MoveL [[1651.97,-191.36,-511.21],[0.032971,0.999448,0.003972,-0.00071],[0,-1,-1,0],[0,9E9,9E9,9E9,9E9,9E9]],Work,z10,custom_tool1\WObj:=WObj0;
MoveL [[1651.88,-186.36,-511.2],[0.032971,0.999448,0.003972,-0.00071],[0,-1,-1,0],[0,9E9,9E9,9E9,9E9,9E9]],Work,z10,custom_tool1\WObj:=WObj0;
MoveL [[1651.8,-181.36,-511.19],[0.032971,0.999448,0.003972,-0.00071],[0,-1,-1,0],[0,9E9,9E9,9E9,9E9,9E9]],Work,z10,custom_tool1\WObj:=WObj0;
MoveL [[1651.72,-176.36,-511.19],[0.032971,0.999448,0.003972,-0.00071],[0,-1,-1,0],[0,9E9,9E9,9E9,9E9,9E9]],Work,z10,custom_tool1\WObj:=WObj0;
MoveL [[1651.64,-171.36,-511.18],[0.032971,0.999448,0.003972,-0.00071],[0,-1,-1,0],[0,9E9,9E9,9E9,9E9,9E9]],Work,z10,custom_tool1\WObj:=WObj0;
MoveL [[1651.55,-166.36,-511.17],[0.032971,0.999448,0.003972,-0.00071],[0,-1,-1,0],[0,9E9,9E9,9E9,9E9,9E9]],Work,z10,custom_tool1\WObj:=WObj0;
MoveL [[1651.47,-161.36,-511.16],[0.032971,0.999448,0.003972,-0.00071],[0,-1,-1,0],[0,9E9,9E9,9E9,9E9,9E9]],Work,z10,custom_tool1\WObj:=WObj0;
MoveL [[1651.39,-156.36,-511.16],[0.032971,0.999448,0.003972,-0.00071],[0,-1,-1,0],[0,9E9,9E9,9E9,9E9,9E9]],Work,z10,custom_tool1\WObj:=WObj0;
MoveL [[1651.31,-151.36,-511.15],[0.032971,0.999448,0.003972,-0.00071],[0,-1,-1,0],[0,9E9,9E9,9E9,9E9,9E9]],Work,z10,custom_tool1\WObj:=WObj0;
MoveL [[1650.68,-145.74,-511.14],[0.032971,0.999448,0.003972,-0.00071],[0,-1,-1,0],[0,9E9,9E9,9E9,9E9,9E9]],Work,z10,custom_tool1\WObj:=WObj0;
MoveL [[1650.05,-140.11,-511.13],[0.032971,0.999448,0.003972,-0.00071],[0,-1,-1,0],[0,9E9,9E9,9E9,9E9,9E9]],Work,z10,custom_tool1\WObj:=WObj0;
MoveL [[1648.24,-134.38,-511.12],[0.032971,0.999448,0.003972,-0.00071],[0,-1,-1,0],[0,9E9,9E9,9E9,9E9,9E9]],Work,z10,custom_tool1\WObj:=WObj0;
MoveL [[1646.43,-128.65,-511.11],[0.032971,0.999448,0.003972,-0.00071],[0,-1,-1,0],[0,9E9,9E9,9E9,9E9,9E9]],Work,z10,custom_tool1\WObj:=WObj0;
MoveL [[1643.51,-123.38,-511.1],[0.032971,0.999448,0.003972,-0.00071],[0,-1,-1,0],[0,9E9,9E9,9E9,9E9,9E9]],Work,z10,custom_tool1\WObj:=WObj0;
MoveL [[1640.59,-118.12,-511.08],[0.032971,0.999448,0.003972,-0.00071],[0,-1,-1,0],[0,9E9,9E9,9E9,9E9,9E9]],Work,z10,custom_tool1\WObj:=WObj0;
MoveL [[1636.59,-113.46,-511.07],[0.032971,0.999448,0.003972,-0.00071],[0,-1,-1,0],[0,9E9,9E9,9E9,9E9,9E9]],Work,z10,custom_tool1\WObj:=WObj0;
MoveL [[1632.58,-108.8,-511.06],[0.032971,0.999448,0.003972,-0.00071],[0,-1,-1,0],[0,9E9,9E9,9E9,9E9,9E9]],Work,z10,custom_tool1\WObj:=WObj0;
MoveL [[1627.75,-105.08,-511.04],[0.032971,0.999448,0.003972,-0.00071],[0,-1,-1,0],[0,9E9,9E9,9E9,9E9,9E9]],Work,z10,custom_tool1\WObj:=WObj0;
MoveL [[1622.92,-101.35,-511.03],[0.032971,0.999448,0.003972,-0.00071],[0,-1,-1,0],[0,9E9,9E9,9E9,9E9,9E9]],Work,z10,custom_tool1\WObj:=WObj0;
MoveL [[1617.56,-98.73,-511.01],[0.032971,0.999448,0.003972,-0.00071],[0,-1,-1,0],[0,9E9,9E9,9E9,9E9,9E9]],Work,z10,custom_tool1\WObj:=WObj0;
MoveL [[1612.2,-96.1,-511],[0.032971,0.999448,0.003972,-0.00071],[0,-1,-1,0],[0,9E9,9E9,9E9,9E9,9E9]],Work,z10,custom_tool1\WObj:=WObj0;
MoveL [[1606.66,-94.63,-510.98],[0.032971,0.999448,0.003972,-0.00071],[0,-1,-1,0],[0,9E9,9E9,9E9,9E9,9E9]],Work,z10,custom_tool1\WObj:=WObj0;
MoveL [[1601.12,-93.16,-510.97],[0.032971,0.999448,0.003972,-0.00071],[0,-1,-1,0],[0,9E9,9E9,9E9,9E9,9E9]],Work,z10,custom_tool1\WObj:=WObj0;
MoveL [[1595.72,-92.76,-510.96],[0.032971,0.999448,0.003972,-0.00071],[0,-1,-1,0],[0,9E9,9E9,9E9,9E9,9E9]],Work,z10,custom_tool1\WObj:=WObj0;
MoveL [[1590.33,-92.36,-510.95],[0.032971,0.999448,0.003972,-0.00071],[0,-1,-1,0],[0,9E9,9E9,9E9,9E9,9E9]],Work,z10,custom_tool1\WObj:=WObj0;
MoveL [[1585.16,-92.45,-510.94],[0.032971,0.999448,0.003972,-0.00071],[0,-1,-1,0],[0,9E9,9E9,9E9,9E9,9E9]],Work,z10,custom_tool1\WObj:=WObj0;
MoveL [[1579.99,-92.53,-510.93],[0.032971,0.999448,0.003972,-0.00071],[0,-1,-1,0],[0,9E9,9E9,9E9,9E9,9E9]],Work,z10,custom_tool1\WObj:=WObj0;
MoveL [[1574.83,-92.62,-510.92],[0.032971,0.999448,0.003972,-0.00071],[0,-1,-1,0],[0,9E9,9E9,9E9,9E9,9E9]],Work,z10,custom_tool1\WObj:=WObj0;
MoveL [[1569.66,-92.7,-510.91],[0.032971,0.999448,0.003972,-0.00071],[0,-1,-1,0],[0,9E9,9E9,9E9,9E9,9E9]],Work,z10,custom_tool1\WObj:=WObj0;
MoveL [[1564.5,-92.79,-510.9],[0.032971,0.999448,0.003972,-0.00071],[0,-1,-1,0],[0,9E9,9E9,9E9,9E9,9E9]],Work,z10,custom_tool1\WObj:=WObj0;
MoveL [[1559.33,-92.87,-510.89],[0.032971,0.999448,0.003972,-0.00071],[0,-1,-1,0],[0,9E9,9E9,9E9,9E9,9E9]],Work,z10,custom_tool1\WObj:=WObj0;
MoveL [[1554.16,-92.96,-510.88],[0.032971,0.999448,0.003972,-0.00071],[0,-1,-1,0],[0,9E9,9E9,9E9,9E9,9E9]],Work,z10,custom_tool1\WObj:=WObj0;
MoveL [[1549,-93.04,-510.87],[0.032971,0.999448,0.003972,-0.00071],[0,-1,-1,0],[0,9E9,9E9,9E9,9E9,9E9]],Work,z10,custom_tool1\WObj:=WObj0;
MoveL [[1543.83,-93.13,-510.86],[0.032971,0.999448,0.003972,-0.00071],[0,-1,-1,0],[0,9E9,9E9,9E9,9E9,9E9]],Work,z10,custom_tool1\WObj:=WObj0;
MoveL [[1538.67,-93.21,-510.85],[0.032971,0.999448,0.003972,-0.00071],[0,-1,-1,0],[0,9E9,9E9,9E9,9E9,9E9]],Work,z10,custom_tool1\WObj:=WObj0;
MoveL [[1533.5,-93.3,-510.84],[0.032971,0.999448,0.003972,-0.00071],[0,-1,-1,0],[0,9E9,9E9,9E9,9E9,9E9]],Work,z10,custom_tool1\WObj:=WObj0;
MoveL [[1528.33,-93.38,-510.83],[0.032971,0.999448,0.003972,-0.00071],[0,-1,-1,0],[0,9E9,9E9,9E9,9E9,9E9]],Work,z10,custom_tool1\WObj:=WObj0;
MoveL [[1523.41,-94.44,-510.82],[0.032971,0.999448,0.003972,-0.00071],[0,-1,-1,0],[0,9E9,9E9,9E9,9E9,9E9]],Work,z10,custom_tool1\WObj:=WObj0;
MoveL [[1518.49,-95.49,-510.81],[0.032971,0.999448,0.003972,-0.00071],[0,-1,-1,0],[0,9E9,9E9,9E9,9E9,9E9]],Work,z10,custom_tool1\WObj:=WObj0;
MoveL [[1513.57,-96.55,-510.8],[0.032971,0.999448,0.003972,-0.00071],[0,-1,-1,0],[0,9E9,9E9,9E9,9E9,9E9]],Work,z10,custom_tool1\WObj:=WObj0;
MoveL [[1508.65,-97.61,-510.79],[0.032971,0.999448,0.003972,-0.00071],[0,-1,-1,0],[0,9E9,9E9,9E9,9E9,9E9]],Work,z10,custom_tool1\WObj:=WObj0;
MoveL [[1505.66,-98.24,-510.79],[0.032971,0.999448,0.003972,-0.00071],[0,-1,-1,0],[0,9E9,9E9,9E9,9E9,9E9]],Work,z10,custom_tool1\WObj:=WObj0;
MoveL [[1501.69,-101,-510.78],[0.032971,0.999448,0.003972,-0.00071],[0,-1,-1,0],[0,9E9,9E9,9E9,9E9,9E9]],Work,z10,custom_tool1\WObj:=WObj0;
MoveL [[1497.72,-103.77,-510.78],[0.032971,0.999448,0.003972,-0.00071],[0,-1,-1,0],[0,9E9,9E9,9E9,9E9,9E9]],Work,z10,custom_tool1\WObj:=WObj0;
MoveL [[1493.75,-106.54,-510.78],[0.032971,0.999448,0.003972,-0.00071],[0,-1,-1,0],[0,9E9,9E9,9E9,9E9,9E9]],Work,z10,custom_tool1\WObj:=WObj0;
MoveL [[1489.77,-109.31,-510.77],[0.032971,0.999448,0.003972,-0.00071],[0,-1,-1,0],[0,9E9,9E9,9E9,9E9,9E9]],Work,z10,custom_tool1\WObj:=WObj0;
MoveL [[1485.8,-112.07,-510.77],[0.032971,0.999448,0.003972,-0.00071],[0,-1,-1,0],[0,9E9,9E9,9E9,9E9,9E9]],Work,z10,custom_tool1\WObj:=WObj0;
MoveL [[1483.26,-116.15,-510.77],[0.032971,0.999448,0.003972,-0.00071],[0,-1,-1,0],[0,9E9,9E9,9E9,9E9,9E9]],Work,z10,custom_tool1\WObj:=WObj0;
MoveL [[1480.71,-120.23,-510.77],[0.032971,0.999448,0.003972,-0.00071],[0,-1,-1,0],[0,9E9,9E9,9E9,9E9,9E9]],Work,z10,custom_tool1\WObj:=WObj0;
MoveL [[1478.17,-124.31,-510.77],[0.032971,0.999448,0.003972,-0.00071],[0,-1,-1,0],[0,9E9,9E9,9E9,9E9,9E9]],Work,z10,custom_tool1\WObj:=WObj0;
MoveL [[1475.63,-128.39,-510.77],[0.032971,0.999448,0.003972,-0.00071],[0,-1,-1,0],[0,9E9,9E9,9E9,9E9,9E9]],Work,z10,custom_tool1\WObj:=WObj0;
MoveL [[1473.08,-132.47,-510.77],[0.032971,0.999448,0.003972,-0.00071],[0,-1,-1,0],[0,9E9,9E9,9E9,9E9,9E9]],Work,z10,custom_tool1\WObj:=WObj0;
MoveL [[1472.58,-135.41,-510.77],[0.032971,0.999448,0.003972,-0.00071],[0,-1,-1,0],[0,9E9,9E9,9E9,9E9,9E9]],Work,z10,custom_tool1\WObj:=WObj0;
MoveL [[1471.76,-140.15,-510.78],[0.032971,0.999448,0.003972,-0.00071],[0,-1,-1,0],[0,9E9,9E9,9E9,9E9,9E9]],Work,z10,custom_tool1\WObj:=WObj0;
MoveL [[1470.95,-144.89,-510.78],[0.032971,0.999448,0.003972,-0.00071],[0,-1,-1,0],[0,9E9,9E9,9E9,9E9,9E9]],Work,z10,custom_tool1\WObj:=WObj0;
MoveL [[1470.14,-149.63,-510.79],[0.032971,0.999448,0.003972,-0.00071],[0,-1,-1,0],[0,9E9,9E9,9E9,9E9,9E9]],Work,z10,custom_tool1\WObj:=WObj0;
MoveL [[1469.33,-154.36,-510.79],[0.032971,0.999448,0.003972,-0.00071],[0,-1,-1,0],[0,9E9,9E9,9E9,9E9,9E9]],Work,z10,custom_tool1\WObj:=WObj0;
MoveL [[1469.41,-159.35,-510.8],[0.032971,0.999448,0.003972,-0.00071],[0,-1,-1,0],[0,9E9,9E9,9E9,9E9,9E9]],Work,z10,custom_tool1\WObj:=WObj0;
MoveL [[1469.5,-164.33,-510.81],[0.032971,0.999448,0.003972,-0.00071],[0,-1,-1,0],[0,9E9,9E9,9E9,9E9,9E9]],Work,z10,custom_tool1\WObj:=WObj0;
MoveL [[1469.58,-169.31,-510.81],[0.032971,0.999448,0.003972,-0.00071],[0,-1,-1,0],[0,9E9,9E9,9E9,9E9,9E9]],Work,z10,custom_tool1\WObj:=WObj0;
MoveL [[1469.66,-174.29,-510.82],[0.032971,0.999448,0.003972,-0.00071],[0,-1,-1,0],[0,9E9,9E9,9E9,9E9,9E9]],Work,z10,custom_tool1\WObj:=WObj0;
MoveL [[1469.74,-179.28,-510.83],[0.032971,0.999448,0.003972,-0.00071],[0,-1,-1,0],[0,9E9,9E9,9E9,9E9,9E9]],Work,z10,custom_tool1\WObj:=WObj0;
MoveL [[1469.82,-184.26,-510.83],[0.032971,0.999448,0.003972,-0.00071],[0,-1,-1,0],[0,9E9,9E9,9E9,9E9,9E9]],Work,z10,custom_tool1\WObj:=WObj0;
MoveL [[1469.91,-189.24,-510.84],[0.032971,0.999448,0.003972,-0.00071],[0,-1,-1,0],[0,9E9,9E9,9E9,9E9,9E9]],Work,z10,custom_tool1\WObj:=WObj0;
MoveL [[1469.99,-194.23,-510.85],[0.032971,0.999448,0.003972,-0.00071],[0,-1,-1,0],[0,9E9,9E9,9E9,9E9,9E9]],Work,z10,custom_tool1\WObj:=WObj0;
MoveL [[1470.07,-199.21,-510.85],[0.032971,0.999448,0.003972,-0.00071],[0,-1,-1,0],[0,9E9,9E9,9E9,9E9,9E9]],Work,z10,custom_tool1\WObj:=WObj0;
MoveL [[1470.15,-204.19,-510.86],[0.032971,0.999448,0.003972,-0.00071],[0,-1,-1,0],[0,9E9,9E9,9E9,9E9,9E9]],Work,z10,custom_tool1\WObj:=WObj0;
MoveL [[1470.24,-209.17,-510.87],[0.032971,0.999448,0.003972,-0.00071],[0,-1,-1,0],[0,9E9,9E9,9E9,9E9,9E9]],Work,z10,custom_tool1\WObj:=WObj0;
MoveL [[1470.32,-214.16,-510.88],[0.032971,0.999448,0.003972,-0.00071],[0,-1,-1,0],[0,9E9,9E9,9E9,9E9,9E9]],Work,z10,custom_tool1\WObj:=WObj0;
MoveL [[1470.4,-219.14,-510.88],[0.032971,0.999448,0.003972,-0.00071],[0,-1,-1,0],[0,9E9,9E9,9E9,9E9,9E9]],Work,z10,custom_tool1\WObj:=WObj0;
MoveL [[1470.48,-224.12,-510.89],[0.032971,0.999448,0.003972,-0.00071],[0,-1,-1,0],[0,9E9,9E9,9E9,9E9,9E9]],Work,z10,custom_tool1\WObj:=WObj0;
MoveL [[1470.56,-229.1,-510.9],[0.032971,0.999448,0.003972,-0.00071],[0,-1,-1,0],[0,9E9,9E9,9E9,9E9,9E9]],Work,z10,custom_tool1\WObj:=WObj0;
MoveL [[1470.65,-234.09,-510.9],[0.032971,0.999448,0.003972,-0.00071],[0,-1,-1,0],[0,9E9,9E9,9E9,9E9,9E9]],Work,z10,custom_tool1\WObj:=WObj0;
MoveL [[1470.73,-239.07,-510.91],[0.032971,0.999448,0.003972,-0.00071],[0,-1,-1,0],[0,9E9,9E9,9E9,9E9,9E9]],Work,z10,custom_tool1\WObj:=WObj0;
MoveL [[1470.81,-244.05,-510.92],[0.032971,0.999448,0.003972,-0.00071],[0,-1,-1,0],[0,9E9,9E9,9E9,9E9,9E9]],Work,z10,custom_tool1\WObj:=WObj0;
MoveL [[1470.89,-249.03,-510.92],[0.032971,0.999448,0.003972,-0.00071],[0,-1,-1,0],[0,9E9,9E9,9E9,9E9,9E9]],Work,z10,custom_tool1\WObj:=WObj0;
MoveL [[1470.97,-254.02,-510.93],[0.032971,0.999448,0.003972,-0.00071],[0,-1,-1,0],[0,9E9,9E9,9E9,9E9,9E9]],Work,z10,custom_tool1\WObj:=WObj0;
MoveL [[1471.06,-259.13,-510.94],[0.032971,0.999448,0.003972,-0.00071],[0,-1,-1,0],[0,9E9,9E9,9E9,9E9,9E9]],Work,z10,custom_tool1\WObj:=WObj0;
MoveL [[1471.14,-264.24,-510.94],[0.032971,0.999448,0.003972,-0.00071],[0,-1,-1,0],[0,9E9,9E9,9E9,9E9,9E9]],Work,z10,custom_tool1\WObj:=WObj0;
MoveL [[1471.23,-269.35,-510.95],[0.032971,0.999448,0.003972,-0.00071],[0,-1,-1,0],[0,9E9,9E9,9E9,9E9,9E9]],Work,z10,custom_tool1\WObj:=WObj0;
MoveL [[1471.31,-274.46,-510.96],[0.032971,0.999448,0.003972,-0.00071],[0,-1,-1,0],[0,9E9,9E9,9E9,9E9,9E9]],Work,z10,custom_tool1\WObj:=WObj0;
MoveL [[1471.4,-279.57,-510.97],[0.032971,0.999448,0.003972,-0.00071],[0,-1,-1,0],[0,9E9,9E9,9E9,9E9,9E9]],Work,z10,custom_tool1\WObj:=WObj0;
MoveL [[1471.48,-284.68,-510.97],[0.032971,0.999448,0.003972,-0.00071],[0,-1,-1,0],[0,9E9,9E9,9E9,9E9,9E9]],Work,z10,custom_tool1\WObj:=WObj0;
MoveL [[1471.56,-289.66,-510.98],[0.032971,0.999448,0.003972,-0.00071],[0,-1,-1,0],[0,9E9,9E9,9E9,9E9,9E9]],Work,z10,custom_tool1\WObj:=WObj0;
MoveL [[1471.64,-294.64,-510.99],[0.032971,0.999448,0.003972,-0.00071],[0,-1,-1,0],[0,9E9,9E9,9E9,9E9,9E9]],Work,z10,custom_tool1\WObj:=WObj0;
MoveL [[1471.73,-299.63,-510.99],[0.032971,0.999448,0.003972,-0.00071],[0,-1,-1,0],[0,9E9,9E9,9E9,9E9,9E9]],Work,z10,custom_tool1\WObj:=WObj0;
MoveL [[1471.81,-304.61,-511],[0.032971,0.999448,0.003972,-0.00071],[0,-1,-1,0],[0,9E9,9E9,9E9,9E9,9E9]],Work,z10,custom_tool1\WObj:=WObj0;
MoveL [[1471.89,-309.59,-511.01],[0.032971,0.999448,0.003972,-0.00071],[0,-1,-1,0],[0,9E9,9E9,9E9,9E9,9E9]],Work,z10,custom_tool1\WObj:=WObj0;
MoveL [[1471.97,-314.58,-511.01],[0.032971,0.999448,0.003972,-0.00071],[0,-1,-1,0],[0,9E9,9E9,9E9,9E9,9E9]],Work,z10,custom_tool1\WObj:=WObj0;
MoveL [[1472.06,-319.56,-511.02],[0.032971,0.999448,0.003972,-0.00071],[0,-1,-1,0],[0,9E9,9E9,9E9,9E9,9E9]],Work,z10,custom_tool1\WObj:=WObj0;
MoveL [[1472.14,-324.54,-511.03],[0.032971,0.999448,0.003972,-0.00071],[0,-1,-1,0],[0,9E9,9E9,9E9,9E9,9E9]],Work,z10,custom_tool1\WObj:=WObj0;
MoveL [[1472.22,-329.52,-511.04],[0.032971,0.999448,0.003972,-0.00071],[0,-1,-1,0],[0,9E9,9E9,9E9,9E9,9E9]],Work,z10,custom_tool1\WObj:=WObj0;
MoveL [[1472.3,-334.51,-511.04],[0.032971,0.999448,0.003972,-0.00071],[0,-1,-1,0],[0,9E9,9E9,9E9,9E9,9E9]],Work,z10,custom_tool1\WObj:=WObj0;
MoveL [[1472.38,-339.49,-511.05],[0.032971,0.999448,0.003972,-0.00071],[0,-1,-1,0],[0,9E9,9E9,9E9,9E9,9E9]],Work,z10,custom_tool1\WObj:=WObj0;
MoveL [[1472.47,-344.47,-511.06],[0.032971,0.999448,0.003972,-0.00071],[0,-1,-1,0],[0,9E9,9E9,9E9,9E9,9E9]],Work,z10,custom_tool1\WObj:=WObj0;
MoveL [[1472.55,-349.45,-511.06],[0.032971,0.999448,0.003972,-0.00071],[0,-1,-1,0],[0,9E9,9E9,9E9,9E9,9E9]],Work,z10,custom_tool1\WObj:=WObj0;
MoveL [[1472.63,-354.44,-511.07],[0.032971,0.999448,0.003972,-0.00071],[0,-1,-1,0],[0,9E9,9E9,9E9,9E9,9E9]],Work,z10,custom_tool1\WObj:=WObj0;
MoveL [[1472.71,-359.42,-511.08],[0.032971,0.999448,0.003972,-0.00071],[0,-1,-1,0],[0,9E9,9E9,9E9,9E9,9E9]],Work,z10,custom_tool1\WObj:=WObj0;
MoveL [[1472.79,-364.4,-511.08],[0.032971,0.999448,0.003972,-0.00071],[0,-1,-1,0],[0,9E9,9E9,9E9,9E9,9E9]],Work,z10,custom_tool1\WObj:=WObj0;
MoveL [[1472.88,-369.38,-511.09],[0.032971,0.999448,0.003972,-0.00071],[0,-1,-1,0],[0,9E9,9E9,9E9,9E9,9E9]],Work,z10,custom_tool1\WObj:=WObj0;
MoveL [[1472.96,-374.37,-511.1],[0.032971,0.999448,0.003972,-0.00071],[0,-1,-1,0],[0,9E9,9E9,9E9,9E9,9E9]],Work,z10,custom_tool1\WObj:=WObj0;
MoveL [[1473.04,-379.35,-511.1],[0.032971,0.999448,0.003972,-0.00071],[0,-1,-1,0],[0,9E9,9E9,9E9,9E9,9E9]],Work,z10,custom_tool1\WObj:=WObj0;
MoveL [[1473.12,-384.33,-511.11],[0.032971,0.999448,0.003972,-0.00071],[0,-1,-1,0],[0,9E9,9E9,9E9,9E9,9E9]],Work,z10,custom_tool1\WObj:=WObj0;
MoveL [[1474.18,-389.25,-511.12],[0.032971,0.999448,0.003972,-0.00071],[0,-1,-1,0],[0,9E9,9E9,9E9,9E9,9E9]],Work,z10,custom_tool1\WObj:=WObj0;
MoveL [[1475.24,-394.18,-511.13],[0.032971,0.999448,0.003972,-0.00071],[0,-1,-1,0],[0,9E9,9E9,9E9,9E9,9E9]],Work,z10,custom_tool1\WObj:=WObj0;
MoveL [[1476.29,-399.1,-511.14],[0.032971,0.999448,0.003972,-0.00071],[0,-1,-1,0],[0,9E9,9E9,9E9,9E9,9E9]],Work,z10,custom_tool1\WObj:=WObj0;
MoveL [[1477.35,-404.02,-511.15],[0.032971,0.999448,0.003972,-0.00071],[0,-1,-1,0],[0,9E9,9E9,9E9,9E9,9E9]],Work,z10,custom_tool1\WObj:=WObj0;
MoveL [[1477.98,-407,-511.15],[0.032971,0.999448,0.003972,-0.00071],[0,-1,-1,0],[0,9E9,9E9,9E9,9E9,9E9]],Work,z10,custom_tool1\WObj:=WObj0;
MoveL [[1480.74,-410.98,-511.16],[0.032971,0.999448,0.003972,-0.00071],[0,-1,-1,0],[0,9E9,9E9,9E9,9E9,9E9]],Work,z10,custom_tool1\WObj:=WObj0;
MoveL [[1483.51,-414.95,-511.17],[0.032971,0.999448,0.003972,-0.00071],[0,-1,-1,0],[0,9E9,9E9,9E9,9E9,9E9]],Work,z10,custom_tool1\WObj:=WObj0;
MoveL [[1486.28,-418.92,-511.18],[0.032971,0.999448,0.003972,-0.00071],[0,-1,-1,0],[0,9E9,9E9,9E9,9E9,9E9]],Work,z10,custom_tool1\WObj:=WObj0;
MoveL [[1489.05,-422.89,-511.2],[0.032971,0.999448,0.003972,-0.00071],[0,-1,-1,0],[0,9E9,9E9,9E9,9E9,9E9]],Work,z10,custom_tool1\WObj:=WObj0;
MoveL [[1491.82,-426.87,-511.21],[0.032971,0.999448,0.003972,-0.00071],[0,-1,-1,0],[0,9E9,9E9,9E9,9E9,9E9]],Work,z10,custom_tool1\WObj:=WObj0;
MoveL [[1495.89,-429.41,-511.22],[0.032971,0.999448,0.003972,-0.00071],[0,-1,-1,0],[0,9E9,9E9,9E9,9E9,9E9]],Work,z10,custom_tool1\WObj:=WObj0;
MoveL [[1499.97,-431.95,-511.23],[0.032971,0.999448,0.003972,-0.00071],[0,-1,-1,0],[0,9E9,9E9,9E9,9E9,9E9]],Work,z10,custom_tool1\WObj:=WObj0;
MoveL [[1504.05,-434.5,-511.24],[0.032971,0.999448,0.003972,-0.00071],[0,-1,-1,0],[0,9E9,9E9,9E9,9E9,9E9]],Work,z10,custom_tool1\WObj:=WObj0;
MoveL [[1508.13,-437.04,-511.25],[0.032971,0.999448,0.003972,-0.00071],[0,-1,-1,0],[0,9E9,9E9,9E9,9E9,9E9]],Work,z10,custom_tool1\WObj:=WObj0;
MoveL [[1512.21,-439.58,-511.26],[0.032971,0.999448,0.003972,-0.00071],[0,-1,-1,0],[0,9E9,9E9,9E9,9E9,9E9]],Work,z10,custom_tool1\WObj:=WObj0;
MoveL [[1515.15,-440.09,-511.27],[0.032971,0.999448,0.003972,-0.00071],[0,-1,-1,0],[0,9E9,9E9,9E9,9E9,9E9]],Work,z10,custom_tool1\WObj:=WObj0;
MoveL [[1519.89,-440.9,-511.28],[0.032971,0.999448,0.003972,-0.00071],[0,-1,-1,0],[0,9E9,9E9,9E9,9E9,9E9]],Work,z10,custom_tool1\WObj:=WObj0;
MoveL [[1524.63,-441.71,-511.29],[0.032971,0.999448,0.003972,-0.00071],[0,-1,-1,0],[0,9E9,9E9,9E9,9E9,9E9]],Work,z10,custom_tool1\WObj:=WObj0;
MoveL [[1529.37,-442.52,-511.3],[0.032971,0.999448,0.003972,-0.00071],[0,-1,-1,0],[0,9E9,9E9,9E9,9E9,9E9]],Work,z10,custom_tool1\WObj:=WObj0;
MoveL [[1534.1,-443.33,-511.31],[0.032971,0.999448,0.003972,-0.00071],[0,-1,-1,0],[0,9E9,9E9,9E9,9E9,9E9]],Work,z10,custom_tool1\WObj:=WObj0;
MoveL [[1539.27,-443.25,-511.32],[0.032971,0.999448,0.003972,-0.00071],[0,-1,-1,0],[0,9E9,9E9,9E9,9E9,9E9]],Work,z10,custom_tool1\WObj:=WObj0;
MoveL [[1544.44,-443.16,-511.33],[0.032971,0.999448,0.003972,-0.00071],[0,-1,-1,0],[0,9E9,9E9,9E9,9E9,9E9]],Work,z10,custom_tool1\WObj:=WObj0;
MoveL [[1549.6,-443.08,-511.34],[0.032971,0.999448,0.003972,-0.00071],[0,-1,-1,0],[0,9E9,9E9,9E9,9E9,9E9]],Work,z10,custom_tool1\WObj:=WObj0;
MoveL [[1554.77,-442.99,-511.35],[0.032971,0.999448,0.003972,-0.00071],[0,-1,-1,0],[0,9E9,9E9,9E9,9E9,9E9]],Work,z10,custom_tool1\WObj:=WObj0;
MoveL [[1559.93,-442.91,-511.36],[0.032971,0.999448,0.003972,-0.00071],[0,-1,-1,0],[0,9E9,9E9,9E9,9E9,9E9]],Work,z10,custom_tool1\WObj:=WObj0;
MoveL [[1565.1,-442.82,-511.37],[0.032971,0.999448,0.003972,-0.00071],[0,-1,-1,0],[0,9E9,9E9,9E9,9E9,9E9]],Work,z10,custom_tool1\WObj:=WObj0;
MoveL [[1570.27,-442.74,-511.38],[0.032971,0.999448,0.003972,-0.00071],[0,-1,-1,0],[0,9E9,9E9,9E9,9E9,9E9]],Work,z10,custom_tool1\WObj:=WObj0;
MoveL [[1575.43,-442.65,-511.39],[0.032971,0.999448,0.003972,-0.00071],[0,-1,-1,0],[0,9E9,9E9,9E9,9E9,9E9]],Work,z10,custom_tool1\WObj:=WObj0;
MoveL [[1580.6,-442.57,-511.41],[0.032971,0.999448,0.003972,-0.00071],[0,-1,-1,0],[0,9E9,9E9,9E9,9E9,9E9]],Work,z10,custom_tool1\WObj:=WObj0;
MoveL [[1585.76,-442.48,-511.42],[0.032971,0.999448,0.003972,-0.00071],[0,-1,-1,0],[0,9E9,9E9,9E9,9E9,9E9]],Work,z10,custom_tool1\WObj:=WObj0;
MoveL [[1590.93,-442.4,-511.43],[0.032971,0.999448,0.003972,-0.00071],[0,-1,-1,0],[0,9E9,9E9,9E9,9E9,9E9]],Work,z10,custom_tool1\WObj:=WObj0;
MoveL [[1596.1,-442.31,-511.44],[0.032971,0.999448,0.003972,-0.00071],[0,-1,-1,0],[0,9E9,9E9,9E9,9E9,9E9]],Work,z10,custom_tool1\WObj:=WObj0;
MoveL [[1601.91,-441.07,-508.45],[0.032971,0.999448,0.003972,-0.00071],[0,-1,-1,0],[0,9E9,9E9,9E9,9E9,9E9]],Work,z10,custom_tool1\WObj:=WObj0;
MoveL [[1607.04,-439.97,-508.45],[0.032971,0.999448,0.003972,-0.00071],[0,-1,-1,0],[0,9E9,9E9,9E9,9E9,9E9]],Work,z10,custom_tool1\WObj:=WObj0;
MoveL [[1612.17,-438.87,-508.46],[0.032971,0.999448,0.003972,-0.00071],[0,-1,-1,0],[0,9E9,9E9,9E9,9E9,9E9]],Work,z10,custom_tool1\WObj:=WObj0;
MoveL [[1617.3,-437.77,-508.47],[0.032971,0.999448,0.003972,-0.00071],[0,-1,-1,0],[0,9E9,9E9,9E9,9E9,9E9]],Work,z10,custom_tool1\WObj:=WObj0;
MoveL [[1618.8,-437.45,-508.47],[0.032971,0.999448,0.003972,-0.00071],[0,-1,-1,0],[0,9E9,9E9,9E9,9E9,9E9]],Work,z10,custom_tool1\WObj:=WObj0;
MoveL [[1622.77,-434.68,-508.48],[0.032971,0.999448,0.003972,-0.00071],[0,-1,-1,0],[0,9E9,9E9,9E9,9E9,9E9]],Work,z10,custom_tool1\WObj:=WObj0;
MoveL [[1626.74,-431.92,-508.48],[0.032971,0.999448,0.003972,-0.00071],[0,-1,-1,0],[0,9E9,9E9,9E9,9E9,9E9]],Work,z10,custom_tool1\WObj:=WObj0;
MoveL [[1630.71,-429.15,-508.49],[0.032971,0.999448,0.003972,-0.00071],[0,-1,-1,0],[0,9E9,9E9,9E9,9E9,9E9]],Work,z10,custom_tool1\WObj:=WObj0;
MoveL [[1634.68,-426.38,-508.49],[0.032971,0.999448,0.003972,-0.00071],[0,-1,-1,0],[0,9E9,9E9,9E9,9E9,9E9]],Work,z10,custom_tool1\WObj:=WObj0;
MoveL [[1638.65,-423.61,-508.5],[0.032971,0.999448,0.003972,-0.00071],[0,-1,-1,0],[0,9E9,9E9,9E9,9E9,9E9]],Work,z10,custom_tool1\WObj:=WObj0;
MoveL [[1641.19,-419.53,-508.49],[0.032971,0.999448,0.003972,-0.00071],[0,-1,-1,0],[0,9E9,9E9,9E9,9E9,9E9]],Work,z10,custom_tool1\WObj:=WObj0;
MoveL [[1643.73,-415.45,-508.49],[0.032971,0.999448,0.003972,-0.00071],[0,-1,-1,0],[0,9E9,9E9,9E9,9E9,9E9]],Work,z10,custom_tool1\WObj:=WObj0;
MoveL [[1646.27,-411.37,-508.49],[0.032971,0.999448,0.003972,-0.00071],[0,-1,-1,0],[0,9E9,9E9,9E9,9E9,9E9]],Work,z10,custom_tool1\WObj:=WObj0;
MoveL [[1648.82,-407.3,-508.49],[0.032971,0.999448,0.003972,-0.00071],[0,-1,-1,0],[0,9E9,9E9,9E9,9E9,9E9]],Work,z10,custom_tool1\WObj:=WObj0;
MoveL [[1651.36,-403.22,-508.49],[0.032971,0.999448,0.003972,-0.00071],[0,-1,-1,0],[0,9E9,9E9,9E9,9E9,9E9]],Work,z10,custom_tool1\WObj:=WObj0;
MoveL [[1651.61,-401.75,-508.49],[0.032971,0.999448,0.003972,-0.00071],[0,-1,-1,0],[0,9E9,9E9,9E9,9E9,9E9]],Work,z10,custom_tool1\WObj:=WObj0;
MoveL [[1652.48,-396.65,-508.49],[0.032971,0.999448,0.003972,-0.00071],[0,-1,-1,0],[0,9E9,9E9,9E9,9E9,9E9]],Work,z10,custom_tool1\WObj:=WObj0;
MoveL [[1653.36,-391.54,-508.48],[0.032971,0.999448,0.003972,-0.00071],[0,-1,-1,0],[0,9E9,9E9,9E9,9E9,9E9]],Work,z10,custom_tool1\WObj:=WObj0;
MoveL [[1654.23,-386.44,-508.48],[0.032971,0.999448,0.003972,-0.00071],[0,-1,-1,0],[0,9E9,9E9,9E9,9E9,9E9]],Work,z10,custom_tool1\WObj:=WObj0;
MoveL [[1655.1,-381.34,-508.47],[0.032971,0.999448,0.003972,-0.00071],[0,-1,-1,0],[0,9E9,9E9,9E9,9E9,9E9]],Work,z10,custom_tool1\WObj:=WObj0;
MoveL [[1655.02,-376.34,-508.46],[0.032971,0.999448,0.003972,-0.00071],[0,-1,-1,0],[0,9E9,9E9,9E9,9E9,9E9]],Work,z10,custom_tool1\WObj:=WObj0;
MoveL [[1654.94,-371.34,-508.46],[0.032971,0.999448,0.003972,-0.00071],[0,-1,-1,0],[0,9E9,9E9,9E9,9E9,9E9]],Work,z10,custom_tool1\WObj:=WObj0;
MoveL [[1654.86,-366.34,-508.45],[0.032971,0.999448,0.003972,-0.00071],[0,-1,-1,0],[0,9E9,9E9,9E9,9E9,9E9]],Work,z10,custom_tool1\WObj:=WObj0;
MoveL [[1654.77,-361.34,-508.44],[0.032971,0.999448,0.003972,-0.00071],[0,-1,-1,0],[0,9E9,9E9,9E9,9E9,9E9]],Work,z10,custom_tool1\WObj:=WObj0;
MoveL [[1654.69,-356.34,-508.44],[0.032971,0.999448,0.003972,-0.00071],[0,-1,-1,0],[0,9E9,9E9,9E9,9E9,9E9]],Work,z10,custom_tool1\WObj:=WObj0;
MoveL [[1654.61,-351.34,-508.43],[0.032971,0.999448,0.003972,-0.00071],[0,-1,-1,0],[0,9E9,9E9,9E9,9E9,9E9]],Work,z10,custom_tool1\WObj:=WObj0;
MoveL [[1654.53,-346.34,-508.42],[0.032971,0.999448,0.003972,-0.00071],[0,-1,-1,0],[0,9E9,9E9,9E9,9E9,9E9]],Work,z10,custom_tool1\WObj:=WObj0;
MoveL [[1654.44,-341.34,-508.41],[0.032971,0.999448,0.003972,-0.00071],[0,-1,-1,0],[0,9E9,9E9,9E9,9E9,9E9]],Work,z10,custom_tool1\WObj:=WObj0;
MoveL [[1654.36,-336.34,-508.41],[0.032971,0.999448,0.003972,-0.00071],[0,-1,-1,0],[0,9E9,9E9,9E9,9E9,9E9]],Work,z10,custom_tool1\WObj:=WObj0;
MoveL [[1654.28,-331.34,-508.4],[0.032971,0.999448,0.003972,-0.00071],[0,-1,-1,0],[0,9E9,9E9,9E9,9E9,9E9]],Work,z10,custom_tool1\WObj:=WObj0;
MoveL [[1654.2,-326.34,-508.39],[0.032971,0.999448,0.003972,-0.00071],[0,-1,-1,0],[0,9E9,9E9,9E9,9E9,9E9]],Work,z10,custom_tool1\WObj:=WObj0;
MoveL [[1654.11,-321.34,-508.39],[0.032971,0.999448,0.003972,-0.00071],[0,-1,-1,0],[0,9E9,9E9,9E9,9E9,9E9]],Work,z10,custom_tool1\WObj:=WObj0;
MoveL [[1654.03,-316.34,-508.38],[0.032971,0.999448,0.003972,-0.00071],[0,-1,-1,0],[0,9E9,9E9,9E9,9E9,9E9]],Work,z10,custom_tool1\WObj:=WObj0;
MoveL [[1653.95,-311.35,-508.37],[0.032971,0.999448,0.003972,-0.00071],[0,-1,-1,0],[0,9E9,9E9,9E9,9E9,9E9]],Work,z10,custom_tool1\WObj:=WObj0;
MoveL [[1653.87,-306.35,-508.37],[0.032971,0.999448,0.003972,-0.00071],[0,-1,-1,0],[0,9E9,9E9,9E9,9E9,9E9]],Work,z10,custom_tool1\WObj:=WObj0;
MoveL [[1653.79,-301.35,-508.36],[0.032971,0.999448,0.003972,-0.00071],[0,-1,-1,0],[0,9E9,9E9,9E9,9E9,9E9]],Work,z10,custom_tool1\WObj:=WObj0;
MoveL [[1653.7,-296.35,-508.35],[0.032971,0.999448,0.003972,-0.00071],[0,-1,-1,0],[0,9E9,9E9,9E9,9E9,9E9]],Work,z10,custom_tool1\WObj:=WObj0;
MoveL [[1653.62,-291.35,-508.35],[0.032971,0.999448,0.003972,-0.00071],[0,-1,-1,0],[0,9E9,9E9,9E9,9E9,9E9]],Work,z10,custom_tool1\WObj:=WObj0;
MoveL [[1653.54,-286.35,-508.34],[0.032971,0.999448,0.003972,-0.00071],[0,-1,-1,0],[0,9E9,9E9,9E9,9E9,9E9]],Work,z10,custom_tool1\WObj:=WObj0;
MoveL [[1653.46,-281.35,-508.33],[0.032971,0.999448,0.003972,-0.00071],[0,-1,-1,0],[0,9E9,9E9,9E9,9E9,9E9]],Work,z10,custom_tool1\WObj:=WObj0;
MoveL [[1653.37,-276.35,-508.32],[0.032971,0.999448,0.003972,-0.00071],[0,-1,-1,0],[0,9E9,9E9,9E9,9E9,9E9]],Work,z10,custom_tool1\WObj:=WObj0;
MoveL [[1653.29,-271.35,-508.32],[0.032971,0.999448,0.003972,-0.00071],[0,-1,-1,0],[0,9E9,9E9,9E9,9E9,9E9]],Work,z10,custom_tool1\WObj:=WObj0;
MoveL [[1653.21,-266.35,-508.31],[0.032971,0.999448,0.003972,-0.00071],[0,-1,-1,0],[0,9E9,9E9,9E9,9E9,9E9]],Work,z10,custom_tool1\WObj:=WObj0;
MoveL [[1653.13,-261.35,-508.3],[0.032971,0.999448,0.003972,-0.00071],[0,-1,-1,0],[0,9E9,9E9,9E9,9E9,9E9]],Work,z10,custom_tool1\WObj:=WObj0;
MoveL [[1653.04,-256.35,-508.3],[0.032971,0.999448,0.003972,-0.00071],[0,-1,-1,0],[0,9E9,9E9,9E9,9E9,9E9]],Work,z10,custom_tool1\WObj:=WObj0;
MoveL [[1652.96,-251.35,-508.29],[0.032971,0.999448,0.003972,-0.00071],[0,-1,-1,0],[0,9E9,9E9,9E9,9E9,9E9]],Work,z10,custom_tool1\WObj:=WObj0;
MoveL [[1652.88,-246.35,-508.28],[0.032971,0.999448,0.003972,-0.00071],[0,-1,-1,0],[0,9E9,9E9,9E9,9E9,9E9]],Work,z10,custom_tool1\WObj:=WObj0;
MoveL [[1652.8,-241.35,-508.28],[0.032971,0.999448,0.003972,-0.00071],[0,-1,-1,0],[0,9E9,9E9,9E9,9E9,9E9]],Work,z10,custom_tool1\WObj:=WObj0;
MoveL [[1652.71,-236.36,-508.27],[0.032971,0.999448,0.003972,-0.00071],[0,-1,-1,0],[0,9E9,9E9,9E9,9E9,9E9]],Work,z10,custom_tool1\WObj:=WObj0;
MoveL [[1652.63,-231.36,-508.26],[0.032971,0.999448,0.003972,-0.00071],[0,-1,-1,0],[0,9E9,9E9,9E9,9E9,9E9]],Work,z10,custom_tool1\WObj:=WObj0;
MoveL [[1652.55,-226.36,-508.25],[0.032971,0.999448,0.003972,-0.00071],[0,-1,-1,0],[0,9E9,9E9,9E9,9E9,9E9]],Work,z10,custom_tool1\WObj:=WObj0;
MoveL [[1652.47,-221.36,-508.25],[0.032971,0.999448,0.003972,-0.00071],[0,-1,-1,0],[0,9E9,9E9,9E9,9E9,9E9]],Work,z10,custom_tool1\WObj:=WObj0;
MoveL [[1652.38,-216.36,-508.24],[0.032971,0.999448,0.003972,-0.00071],[0,-1,-1,0],[0,9E9,9E9,9E9,9E9,9E9]],Work,z10,custom_tool1\WObj:=WObj0;
MoveL [[1652.3,-211.36,-508.23],[0.032971,0.999448,0.003972,-0.00071],[0,-1,-1,0],[0,9E9,9E9,9E9,9E9,9E9]],Work,z10,custom_tool1\WObj:=WObj0;
MoveL [[1652.22,-206.36,-508.23],[0.032971,0.999448,0.003972,-0.00071],[0,-1,-1,0],[0,9E9,9E9,9E9,9E9,9E9]],Work,z10,custom_tool1\WObj:=WObj0;
MoveL [[1652.14,-201.36,-508.22],[0.032971,0.999448,0.003972,-0.00071],[0,-1,-1,0],[0,9E9,9E9,9E9,9E9,9E9]],Work,z10,custom_tool1\WObj:=WObj0;
MoveL [[1652.05,-196.36,-508.21],[0.032971,0.999448,0.003972,-0.00071],[0,-1,-1,0],[0,9E9,9E9,9E9,9E9,9E9]],Work,z10,custom_tool1\WObj:=WObj0;
MoveL [[1651.97,-191.36,-508.21],[0.032971,0.999448,0.003972,-0.00071],[0,-1,-1,0],[0,9E9,9E9,9E9,9E9,9E9]],Work,z10,custom_tool1\WObj:=WObj0;
MoveL [[1651.89,-186.36,-508.2],[0.032971,0.999448,0.003972,-0.00071],[0,-1,-1,0],[0,9E9,9E9,9E9,9E9,9E9]],Work,z10,custom_tool1\WObj:=WObj0;
MoveL [[1651.81,-181.36,-508.19],[0.032971,0.999448,0.003972,-0.00071],[0,-1,-1,0],[0,9E9,9E9,9E9,9E9,9E9]],Work,z10,custom_tool1\WObj:=WObj0;
MoveL [[1651.72,-176.36,-508.19],[0.032971,0.999448,0.003972,-0.00071],[0,-1,-1,0],[0,9E9,9E9,9E9,9E9,9E9]],Work,z10,custom_tool1\WObj:=WObj0;
MoveL [[1651.64,-171.36,-508.18],[0.032971,0.999448,0.003972,-0.00071],[0,-1,-1,0],[0,9E9,9E9,9E9,9E9,9E9]],Work,z10,custom_tool1\WObj:=WObj0;
MoveL [[1651.56,-166.37,-508.17],[0.032971,0.999448,0.003972,-0.00071],[0,-1,-1,0],[0,9E9,9E9,9E9,9E9,9E9]],Work,z10,custom_tool1\WObj:=WObj0;
MoveL [[1651.48,-161.37,-508.16],[0.032971,0.999448,0.003972,-0.00071],[0,-1,-1,0],[0,9E9,9E9,9E9,9E9,9E9]],Work,z10,custom_tool1\WObj:=WObj0;
MoveL [[1651.39,-156.37,-508.16],[0.032971,0.999448,0.003972,-0.00071],[0,-1,-1,0],[0,9E9,9E9,9E9,9E9,9E9]],Work,z10,custom_tool1\WObj:=WObj0;
MoveL [[1651.31,-151.37,-508.15],[0.032971,0.999448,0.003972,-0.00071],[0,-1,-1,0],[0,9E9,9E9,9E9,9E9,9E9]],Work,z10,custom_tool1\WObj:=WObj0;
MoveL [[1650.69,-145.74,-508.14],[0.032971,0.999448,0.003972,-0.00071],[0,-1,-1,0],[0,9E9,9E9,9E9,9E9,9E9]],Work,z10,custom_tool1\WObj:=WObj0;
MoveL [[1650.06,-140.11,-508.13],[0.032971,0.999448,0.003972,-0.00071],[0,-1,-1,0],[0,9E9,9E9,9E9,9E9,9E9]],Work,z10,custom_tool1\WObj:=WObj0;
MoveL [[1648.25,-134.38,-508.12],[0.032971,0.999448,0.003972,-0.00071],[0,-1,-1,0],[0,9E9,9E9,9E9,9E9,9E9]],Work,z10,custom_tool1\WObj:=WObj0;
MoveL [[1646.44,-128.65,-508.11],[0.032971,0.999448,0.003972,-0.00071],[0,-1,-1,0],[0,9E9,9E9,9E9,9E9,9E9]],Work,z10,custom_tool1\WObj:=WObj0;
MoveL [[1643.52,-123.39,-508.1],[0.032971,0.999448,0.003972,-0.00071],[0,-1,-1,0],[0,9E9,9E9,9E9,9E9,9E9]],Work,z10,custom_tool1\WObj:=WObj0;
MoveL [[1640.59,-118.12,-508.08],[0.032971,0.999448,0.003972,-0.00071],[0,-1,-1,0],[0,9E9,9E9,9E9,9E9,9E9]],Work,z10,custom_tool1\WObj:=WObj0;
MoveL [[1636.59,-113.46,-508.07],[0.032971,0.999448,0.003972,-0.00071],[0,-1,-1,0],[0,9E9,9E9,9E9,9E9,9E9]],Work,z10,custom_tool1\WObj:=WObj0;
MoveL [[1632.59,-108.8,-508.06],[0.032971,0.999448,0.003972,-0.00071],[0,-1,-1,0],[0,9E9,9E9,9E9,9E9,9E9]],Work,z10,custom_tool1\WObj:=WObj0;
MoveL [[1627.76,-105.08,-508.04],[0.032971,0.999448,0.003972,-0.00071],[0,-1,-1,0],[0,9E9,9E9,9E9,9E9,9E9]],Work,z10,custom_tool1\WObj:=WObj0;
MoveL [[1622.93,-101.36,-508.03],[0.032971,0.999448,0.003972,-0.00071],[0,-1,-1,0],[0,9E9,9E9,9E9,9E9,9E9]],Work,z10,custom_tool1\WObj:=WObj0;
MoveL [[1617.57,-98.73,-508.01],[0.032971,0.999448,0.003972,-0.00071],[0,-1,-1,0],[0,9E9,9E9,9E9,9E9,9E9]],Work,z10,custom_tool1\WObj:=WObj0;
MoveL [[1612.2,-96.11,-508],[0.032971,0.999448,0.003972,-0.00071],[0,-1,-1,0],[0,9E9,9E9,9E9,9E9,9E9]],Work,z10,custom_tool1\WObj:=WObj0;
MoveL [[1606.66,-94.64,-507.98],[0.032971,0.999448,0.003972,-0.00071],[0,-1,-1,0],[0,9E9,9E9,9E9,9E9,9E9]],Work,z10,custom_tool1\WObj:=WObj0;
MoveL [[1601.12,-93.16,-507.97],[0.032971,0.999448,0.003972,-0.00071],[0,-1,-1,0],[0,9E9,9E9,9E9,9E9,9E9]],Work,z10,custom_tool1\WObj:=WObj0;
MoveL [[1595.73,-92.76,-507.96],[0.032971,0.999448,0.003972,-0.00071],[0,-1,-1,0],[0,9E9,9E9,9E9,9E9,9E9]],Work,z10,custom_tool1\WObj:=WObj0;
MoveL [[1590.33,-92.36,-507.95],[0.032971,0.999448,0.003972,-0.00071],[0,-1,-1,0],[0,9E9,9E9,9E9,9E9,9E9]],Work,z10,custom_tool1\WObj:=WObj0;
MoveL [[1585.17,-92.45,-507.94],[0.032971,0.999448,0.003972,-0.00071],[0,-1,-1,0],[0,9E9,9E9,9E9,9E9,9E9]],Work,z10,custom_tool1\WObj:=WObj0;
MoveL [[1580,-92.54,-507.93],[0.032971,0.999448,0.003972,-0.00071],[0,-1,-1,0],[0,9E9,9E9,9E9,9E9,9E9]],Work,z10,custom_tool1\WObj:=WObj0;
MoveL [[1574.83,-92.62,-507.92],[0.032971,0.999448,0.003972,-0.00071],[0,-1,-1,0],[0,9E9,9E9,9E9,9E9,9E9]],Work,z10,custom_tool1\WObj:=WObj0;
MoveL [[1569.67,-92.71,-507.91],[0.032971,0.999448,0.003972,-0.00071],[0,-1,-1,0],[0,9E9,9E9,9E9,9E9,9E9]],Work,z10,custom_tool1\WObj:=WObj0;
MoveL [[1564.5,-92.79,-507.9],[0.032971,0.999448,0.003972,-0.00071],[0,-1,-1,0],[0,9E9,9E9,9E9,9E9,9E9]],Work,z10,custom_tool1\WObj:=WObj0;
MoveL [[1559.34,-92.88,-507.89],[0.032971,0.999448,0.003972,-0.00071],[0,-1,-1,0],[0,9E9,9E9,9E9,9E9,9E9]],Work,z10,custom_tool1\WObj:=WObj0;
MoveL [[1554.17,-92.96,-507.88],[0.032971,0.999448,0.003972,-0.00071],[0,-1,-1,0],[0,9E9,9E9,9E9,9E9,9E9]],Work,z10,custom_tool1\WObj:=WObj0;
MoveL [[1549,-93.05,-507.87],[0.032971,0.999448,0.003972,-0.00071],[0,-1,-1,0],[0,9E9,9E9,9E9,9E9,9E9]],Work,z10,custom_tool1\WObj:=WObj0;
MoveL [[1543.84,-93.13,-507.86],[0.032971,0.999448,0.003972,-0.00071],[0,-1,-1,0],[0,9E9,9E9,9E9,9E9,9E9]],Work,z10,custom_tool1\WObj:=WObj0;
MoveL [[1538.67,-93.22,-507.85],[0.032971,0.999448,0.003972,-0.00071],[0,-1,-1,0],[0,9E9,9E9,9E9,9E9,9E9]],Work,z10,custom_tool1\WObj:=WObj0;
MoveL [[1533.51,-93.3,-507.84],[0.032971,0.999448,0.003972,-0.00071],[0,-1,-1,0],[0,9E9,9E9,9E9,9E9,9E9]],Work,z10,custom_tool1\WObj:=WObj0;
MoveL [[1528.34,-93.39,-507.83],[0.032971,0.999448,0.003972,-0.00071],[0,-1,-1,0],[0,9E9,9E9,9E9,9E9,9E9]],Work,z10,custom_tool1\WObj:=WObj0;
MoveL [[1523.04,-94.52,-507.82],[0.032971,0.999448,0.003972,-0.00071],[0,-1,-1,0],[0,9E9,9E9,9E9,9E9,9E9]],Work,z10,custom_tool1\WObj:=WObj0;
MoveL [[1517.74,-95.66,-507.81],[0.032971,0.999448,0.003972,-0.00071],[0,-1,-1,0],[0,9E9,9E9,9E9,9E9,9E9]],Work,z10,custom_tool1\WObj:=WObj0;
MoveL [[1512.44,-96.8,-507.8],[0.032971,0.999448,0.003972,-0.00071],[0,-1,-1,0],[0,9E9,9E9,9E9,9E9,9E9]],Work,z10,custom_tool1\WObj:=WObj0;
MoveL [[1507.14,-97.94,-507.79],[0.032971,0.999448,0.003972,-0.00071],[0,-1,-1,0],[0,9E9,9E9,9E9,9E9,9E9]],Work,z10,custom_tool1\WObj:=WObj0;
MoveL [[1505.65,-98.25,-507.79],[0.032971,0.999448,0.003972,-0.00071],[0,-1,-1,0],[0,9E9,9E9,9E9,9E9,9E9]],Work,z10,custom_tool1\WObj:=WObj0;
MoveL [[1501.68,-101.02,-507.78],[0.032971,0.999448,0.003972,-0.00071],[0,-1,-1,0],[0,9E9,9E9,9E9,9E9,9E9]],Work,z10,custom_tool1\WObj:=WObj0;
MoveL [[1497.7,-103.79,-507.78],[0.032971,0.999448,0.003972,-0.00071],[0,-1,-1,0],[0,9E9,9E9,9E9,9E9,9E9]],Work,z10,custom_tool1\WObj:=WObj0;
MoveL [[1493.73,-106.56,-507.78],[0.032971,0.999448,0.003972,-0.00071],[0,-1,-1,0],[0,9E9,9E9,9E9,9E9,9E9]],Work,z10,custom_tool1\WObj:=WObj0;
MoveL [[1489.76,-109.33,-507.77],[0.032971,0.999448,0.003972,-0.00071],[0,-1,-1,0],[0,9E9,9E9,9E9,9E9,9E9]],Work,z10,custom_tool1\WObj:=WObj0;
MoveL [[1485.79,-112.09,-507.77],[0.032971,0.999448,0.003972,-0.00071],[0,-1,-1,0],[0,9E9,9E9,9E9,9E9,9E9]],Work,z10,custom_tool1\WObj:=WObj0;
MoveL [[1483.25,-116.17,-507.77],[0.032971,0.999448,0.003972,-0.00071],[0,-1,-1,0],[0,9E9,9E9,9E9,9E9,9E9]],Work,z10,custom_tool1\WObj:=WObj0;
MoveL [[1480.71,-120.25,-507.77],[0.032971,0.999448,0.003972,-0.00071],[0,-1,-1,0],[0,9E9,9E9,9E9,9E9,9E9]],Work,z10,custom_tool1\WObj:=WObj0;
MoveL [[1478.17,-124.33,-507.77],[0.032971,0.999448,0.003972,-0.00071],[0,-1,-1,0],[0,9E9,9E9,9E9,9E9,9E9]],Work,z10,custom_tool1\WObj:=WObj0;
MoveL [[1475.63,-128.41,-507.77],[0.032971,0.999448,0.003972,-0.00071],[0,-1,-1,0],[0,9E9,9E9,9E9,9E9,9E9]],Work,z10,custom_tool1\WObj:=WObj0;
MoveL [[1473.08,-132.49,-507.77],[0.032971,0.999448,0.003972,-0.00071],[0,-1,-1,0],[0,9E9,9E9,9E9,9E9,9E9]],Work,z10,custom_tool1\WObj:=WObj0;
MoveL [[1472.83,-133.95,-507.77],[0.032971,0.999448,0.003972,-0.00071],[0,-1,-1,0],[0,9E9,9E9,9E9,9E9,9E9]],Work,z10,custom_tool1\WObj:=WObj0;
MoveL [[1471.96,-139.06,-507.78],[0.032971,0.999448,0.003972,-0.00071],[0,-1,-1,0],[0,9E9,9E9,9E9,9E9,9E9]],Work,z10,custom_tool1\WObj:=WObj0;
MoveL [[1471.08,-144.16,-507.78],[0.032971,0.999448,0.003972,-0.00071],[0,-1,-1,0],[0,9E9,9E9,9E9,9E9,9E9]],Work,z10,custom_tool1\WObj:=WObj0;
MoveL [[1470.21,-149.26,-507.79],[0.032971,0.999448,0.003972,-0.00071],[0,-1,-1,0],[0,9E9,9E9,9E9,9E9,9E9]],Work,z10,custom_tool1\WObj:=WObj0;
MoveL [[1469.34,-154.37,-507.79],[0.032971,0.999448,0.003972,-0.00071],[0,-1,-1,0],[0,9E9,9E9,9E9,9E9,9E9]],Work,z10,custom_tool1\WObj:=WObj0;
MoveL [[1469.42,-159.48,-507.8],[0.032971,0.999448,0.003972,-0.00071],[0,-1,-1,0],[0,9E9,9E9,9E9,9E9,9E9]],Work,z10,custom_tool1\WObj:=WObj0;
MoveL [[1469.51,-164.59,-507.81],[0.032971,0.999448,0.003972,-0.00071],[0,-1,-1,0],[0,9E9,9E9,9E9,9E9,9E9]],Work,z10,custom_tool1\WObj:=WObj0;
MoveL [[1469.59,-169.7,-507.81],[0.032971,0.999448,0.003972,-0.00071],[0,-1,-1,0],[0,9E9,9E9,9E9,9E9,9E9]],Work,z10,custom_tool1\WObj:=WObj0;
MoveL [[1469.67,-174.81,-507.82],[0.032971,0.999448,0.003972,-0.00071],[0,-1,-1,0],[0,9E9,9E9,9E9,9E9,9E9]],Work,z10,custom_tool1\WObj:=WObj0;
MoveL [[1469.76,-179.92,-507.83],[0.032971,0.999448,0.003972,-0.00071],[0,-1,-1,0],[0,9E9,9E9,9E9,9E9,9E9]],Work,z10,custom_tool1\WObj:=WObj0;
MoveL [[1469.84,-185.03,-507.83],[0.032971,0.999448,0.003972,-0.00071],[0,-1,-1,0],[0,9E9,9E9,9E9,9E9,9E9]],Work,z10,custom_tool1\WObj:=WObj0;
MoveL [[1469.93,-190.14,-507.84],[0.032971,0.999448,0.003972,-0.00071],[0,-1,-1,0],[0,9E9,9E9,9E9,9E9,9E9]],Work,z10,custom_tool1\WObj:=WObj0;
MoveL [[1470.01,-195.25,-507.85],[0.032971,0.999448,0.003972,-0.00071],[0,-1,-1,0],[0,9E9,9E9,9E9,9E9,9E9]],Work,z10,custom_tool1\WObj:=WObj0;
MoveL [[1470.1,-200.36,-507.86],[0.032971,0.999448,0.003972,-0.00071],[0,-1,-1,0],[0,9E9,9E9,9E9,9E9,9E9]],Work,z10,custom_tool1\WObj:=WObj0;
MoveL [[1470.18,-205.47,-507.86],[0.032971,0.999448,0.003972,-0.00071],[0,-1,-1,0],[0,9E9,9E9,9E9,9E9,9E9]],Work,z10,custom_tool1\WObj:=WObj0;
MoveL [[1470.26,-210.58,-507.87],[0.032971,0.999448,0.003972,-0.00071],[0,-1,-1,0],[0,9E9,9E9,9E9,9E9,9E9]],Work,z10,custom_tool1\WObj:=WObj0;
MoveL [[1470.35,-215.69,-507.88],[0.032971,0.999448,0.003972,-0.00071],[0,-1,-1,0],[0,9E9,9E9,9E9,9E9,9E9]],Work,z10,custom_tool1\WObj:=WObj0;
MoveL [[1470.43,-220.8,-507.88],[0.032971,0.999448,0.003972,-0.00071],[0,-1,-1,0],[0,9E9,9E9,9E9,9E9,9E9]],Work,z10,custom_tool1\WObj:=WObj0;
MoveL [[1470.52,-225.91,-507.89],[0.032971,0.999448,0.003972,-0.00071],[0,-1,-1,0],[0,9E9,9E9,9E9,9E9,9E9]],Work,z10,custom_tool1\WObj:=WObj0;
MoveL [[1470.6,-231.02,-507.9],[0.032971,0.999448,0.003972,-0.00071],[0,-1,-1,0],[0,9E9,9E9,9E9,9E9,9E9]],Work,z10,custom_tool1\WObj:=WObj0;
MoveL [[1470.69,-236.13,-507.91],[0.032971,0.999448,0.003972,-0.00071],[0,-1,-1,0],[0,9E9,9E9,9E9,9E9,9E9]],Work,z10,custom_tool1\WObj:=WObj0;
MoveL [[1470.77,-241.24,-507.91],[0.032971,0.999448,0.003972,-0.00071],[0,-1,-1,0],[0,9E9,9E9,9E9,9E9,9E9]],Work,z10,custom_tool1\WObj:=WObj0;
MoveL [[1470.85,-246.36,-507.92],[0.032971,0.999448,0.003972,-0.00071],[0,-1,-1,0],[0,9E9,9E9,9E9,9E9,9E9]],Work,z10,custom_tool1\WObj:=WObj0;
MoveL [[1470.94,-251.47,-507.93],[0.032971,0.999448,0.003972,-0.00071],[0,-1,-1,0],[0,9E9,9E9,9E9,9E9,9E9]],Work,z10,custom_tool1\WObj:=WObj0;
MoveL [[1471.02,-256.58,-507.93],[0.032971,0.999448,0.003972,-0.00071],[0,-1,-1,0],[0,9E9,9E9,9E9,9E9,9E9]],Work,z10,custom_tool1\WObj:=WObj0;
MoveL [[1471.11,-261.69,-507.94],[0.032971,0.999448,0.003972,-0.00071],[0,-1,-1,0],[0,9E9,9E9,9E9,9E9,9E9]],Work,z10,custom_tool1\WObj:=WObj0;
MoveL [[1471.19,-266.8,-507.95],[0.032971,0.999448,0.003972,-0.00071],[0,-1,-1,0],[0,9E9,9E9,9E9,9E9,9E9]],Work,z10,custom_tool1\WObj:=WObj0;
MoveL [[1471.28,-271.91,-507.96],[0.032971,0.999448,0.003972,-0.00071],[0,-1,-1,0],[0,9E9,9E9,9E9,9E9,9E9]],Work,z10,custom_tool1\WObj:=WObj0;
MoveL [[1471.36,-277.02,-507.96],[0.032971,0.999448,0.003972,-0.00071],[0,-1,-1,0],[0,9E9,9E9,9E9,9E9,9E9]],Work,z10,custom_tool1\WObj:=WObj0;
MoveL [[1471.44,-282.13,-507.97],[0.032971,0.999448,0.003972,-0.00071],[0,-1,-1,0],[0,9E9,9E9,9E9,9E9,9E9]],Work,z10,custom_tool1\WObj:=WObj0;
MoveL [[1471.53,-287.24,-507.98],[0.032971,0.999448,0.003972,-0.00071],[0,-1,-1,0],[0,9E9,9E9,9E9,9E9,9E9]],Work,z10,custom_tool1\WObj:=WObj0;
MoveL [[1471.61,-292.35,-507.98],[0.032971,0.999448,0.003972,-0.00071],[0,-1,-1,0],[0,9E9,9E9,9E9,9E9,9E9]],Work,z10,custom_tool1\WObj:=WObj0;
MoveL [[1471.7,-297.46,-507.99],[0.032971,0.999448,0.003972,-0.00071],[0,-1,-1,0],[0,9E9,9E9,9E9,9E9,9E9]],Work,z10,custom_tool1\WObj:=WObj0;
MoveL [[1471.78,-302.57,-508],[0.032971,0.999448,0.003972,-0.00071],[0,-1,-1,0],[0,9E9,9E9,9E9,9E9,9E9]],Work,z10,custom_tool1\WObj:=WObj0;
MoveL [[1471.87,-307.68,-508.01],[0.032971,0.999448,0.003972,-0.00071],[0,-1,-1,0],[0,9E9,9E9,9E9,9E9,9E9]],Work,z10,custom_tool1\WObj:=WObj0;
MoveL [[1471.95,-312.79,-508.01],[0.032971,0.999448,0.003972,-0.00071],[0,-1,-1,0],[0,9E9,9E9,9E9,9E9,9E9]],Work,z10,custom_tool1\WObj:=WObj0;
MoveL [[1472.03,-317.9,-508.02],[0.032971,0.999448,0.003972,-0.00071],[0,-1,-1,0],[0,9E9,9E9,9E9,9E9,9E9]],Work,z10,custom_tool1\WObj:=WObj0;
MoveL [[1472.12,-323.01,-508.03],[0.032971,0.999448,0.003972,-0.00071],[0,-1,-1,0],[0,9E9,9E9,9E9,9E9,9E9]],Work,z10,custom_tool1\WObj:=WObj0;
MoveL [[1472.2,-328.12,-508.03],[0.032971,0.999448,0.003972,-0.00071],[0,-1,-1,0],[0,9E9,9E9,9E9,9E9,9E9]],Work,z10,custom_tool1\WObj:=WObj0;
MoveL [[1472.29,-333.23,-508.04],[0.032971,0.999448,0.003972,-0.00071],[0,-1,-1,0],[0,9E9,9E9,9E9,9E9,9E9]],Work,z10,custom_tool1\WObj:=WObj0;
MoveL [[1472.37,-338.34,-508.05],[0.032971,0.999448,0.003972,-0.00071],[0,-1,-1,0],[0,9E9,9E9,9E9,9E9,9E9]],Work,z10,custom_tool1\WObj:=WObj0;
MoveL [[1472.46,-343.45,-508.05],[0.032971,0.999448,0.003972,-0.00071],[0,-1,-1,0],[0,9E9,9E9,9E9,9E9,9E9]],Work,z10,custom_tool1\WObj:=WObj0;
MoveL [[1472.54,-348.56,-508.06],[0.032971,0.999448,0.003972,-0.00071],[0,-1,-1,0],[0,9E9,9E9,9E9,9E9,9E9]],Work,z10,custom_tool1\WObj:=WObj0;
MoveL [[1472.62,-353.67,-508.07],[0.032971,0.999448,0.003972,-0.00071],[0,-1,-1,0],[0,9E9,9E9,9E9,9E9,9E9]],Work,z10,custom_tool1\WObj:=WObj0;
MoveL [[1472.71,-358.78,-508.08],[0.032971,0.999448,0.003972,-0.00071],[0,-1,-1,0],[0,9E9,9E9,9E9,9E9,9E9]],Work,z10,custom_tool1\WObj:=WObj0;
MoveL [[1472.79,-363.89,-508.08],[0.032971,0.999448,0.003972,-0.00071],[0,-1,-1,0],[0,9E9,9E9,9E9,9E9,9E9]],Work,z10,custom_tool1\WObj:=WObj0;
MoveL [[1472.88,-369.01,-508.09],[0.032971,0.999448,0.003972,-0.00071],[0,-1,-1,0],[0,9E9,9E9,9E9,9E9,9E9]],Work,z10,custom_tool1\WObj:=WObj0;
MoveL [[1472.96,-374.12,-508.1],[0.032971,0.999448,0.003972,-0.00071],[0,-1,-1,0],[0,9E9,9E9,9E9,9E9,9E9]],Work,z10,custom_tool1\WObj:=WObj0;
MoveL [[1473.04,-379.23,-508.1],[0.032971,0.999448,0.003972,-0.00071],[0,-1,-1,0],[0,9E9,9E9,9E9,9E9,9E9]],Work,z10,custom_tool1\WObj:=WObj0;
MoveL [[1473.13,-384.34,-508.11],[0.032971,0.999448,0.003972,-0.00071],[0,-1,-1,0],[0,9E9,9E9,9E9,9E9,9E9]],Work,z10,custom_tool1\WObj:=WObj0;
MoveL [[1474.27,-389.64,-508.12],[0.032971,0.999448,0.003972,-0.00071],[0,-1,-1,0],[0,9E9,9E9,9E9,9E9,9E9]],Work,z10,custom_tool1\WObj:=WObj0;
MoveL [[1475.4,-394.94,-508.13],[0.032971,0.999448,0.003972,-0.00071],[0,-1,-1,0],[0,9E9,9E9,9E9,9E9,9E9]],Work,z10,custom_tool1\WObj:=WObj0;
MoveL [[1476.54,-400.24,-508.14],[0.032971,0.999448,0.003972,-0.00071],[0,-1,-1,0],[0,9E9,9E9,9E9,9E9,9E9]],Work,z10,custom_tool1\WObj:=WObj0;
MoveL [[1477.68,-405.54,-508.15],[0.032971,0.999448,0.003972,-0.00071],[0,-1,-1,0],[0,9E9,9E9,9E9,9E9,9E9]],Work,z10,custom_tool1\WObj:=WObj0;
MoveL [[1477.99,-407.03,-508.15],[0.032971,0.999448,0.003972,-0.00071],[0,-1,-1,0],[0,9E9,9E9,9E9,9E9,9E9]],Work,z10,custom_tool1\WObj:=WObj0;
MoveL [[1480.76,-411,-508.16],[0.032971,0.999448,0.003972,-0.00071],[0,-1,-1,0],[0,9E9,9E9,9E9,9E9,9E9]],Work,z10,custom_tool1\WObj:=WObj0;
MoveL [[1483.53,-414.97,-508.17],[0.032971,0.999448,0.003972,-0.00071],[0,-1,-1,0],[0,9E9,9E9,9E9,9E9,9E9]],Work,z10,custom_tool1\WObj:=WObj0;
MoveL [[1486.3,-418.94,-508.19],[0.032971,0.999448,0.003972,-0.00071],[0,-1,-1,0],[0,9E9,9E9,9E9,9E9,9E9]],Work,z10,custom_tool1\WObj:=WObj0;
MoveL [[1489.07,-422.91,-508.2],[0.032971,0.999448,0.003972,-0.00071],[0,-1,-1,0],[0,9E9,9E9,9E9,9E9,9E9]],Work,z10,custom_tool1\WObj:=WObj0;
MoveL [[1491.84,-426.89,-508.21],[0.032971,0.999448,0.003972,-0.00071],[0,-1,-1,0],[0,9E9,9E9,9E9,9E9,9E9]],Work,z10,custom_tool1\WObj:=WObj0;
MoveL [[1495.91,-429.43,-508.22],[0.032971,0.999448,0.003972,-0.00071],[0,-1,-1,0],[0,9E9,9E9,9E9,9E9,9E9]],Work,z10,custom_tool1\WObj:=WObj0;
MoveL [[1499.99,-431.97,-508.23],[0.032971,0.999448,0.003972,-0.00071],[0,-1,-1,0],[0,9E9,9E9,9E9,9E9,9E9]],Work,z10,custom_tool1\WObj:=WObj0;
MoveL [[1504.07,-434.51,-508.24],[0.032971,0.999448,0.003972,-0.00071],[0,-1,-1,0],[0,9E9,9E9,9E9,9E9,9E9]],Work,z10,custom_tool1\WObj:=WObj0;
MoveL [[1508.15,-437.05,-508.25],[0.032971,0.999448,0.003972,-0.00071],[0,-1,-1,0],[0,9E9,9E9,9E9,9E9,9E9]],Work,z10,custom_tool1\WObj:=WObj0;
MoveL [[1512.23,-439.59,-508.26],[0.032971,0.999448,0.003972,-0.00071],[0,-1,-1,0],[0,9E9,9E9,9E9,9E9,9E9]],Work,z10,custom_tool1\WObj:=WObj0;
MoveL [[1513.7,-439.85,-508.27],[0.032971,0.999448,0.003972,-0.00071],[0,-1,-1,0],[0,9E9,9E9,9E9,9E9,9E9]],Work,z10,custom_tool1\WObj:=WObj0;
MoveL [[1518.8,-440.72,-508.28],[0.032971,0.999448,0.003972,-0.00071],[0,-1,-1,0],[0,9E9,9E9,9E9,9E9,9E9]],Work,z10,custom_tool1\WObj:=WObj0;
MoveL [[1523.9,-441.59,-508.29],[0.032971,0.999448,0.003972,-0.00071],[0,-1,-1,0],[0,9E9,9E9,9E9,9E9,9E9]],Work,z10,custom_tool1\WObj:=WObj0;
MoveL [[1529.01,-442.47,-508.3],[0.032971,0.999448,0.003972,-0.00071],[0,-1,-1,0],[0,9E9,9E9,9E9,9E9,9E9]],Work,z10,custom_tool1\WObj:=WObj0;
MoveL [[1534.11,-443.34,-508.31],[0.032971,0.999448,0.003972,-0.00071],[0,-1,-1,0],[0,9E9,9E9,9E9,9E9,9E9]],Work,z10,custom_tool1\WObj:=WObj0;
MoveL [[1539.28,-443.25,-508.32],[0.032971,0.999448,0.003972,-0.00071],[0,-1,-1,0],[0,9E9,9E9,9E9,9E9,9E9]],Work,z10,custom_tool1\WObj:=WObj0;
MoveL [[1544.44,-443.17,-508.33],[0.032971,0.999448,0.003972,-0.00071],[0,-1,-1,0],[0,9E9,9E9,9E9,9E9,9E9]],Work,z10,custom_tool1\WObj:=WObj0;
MoveL [[1549.61,-443.08,-508.34],[0.032971,0.999448,0.003972,-0.00071],[0,-1,-1,0],[0,9E9,9E9,9E9,9E9,9E9]],Work,z10,custom_tool1\WObj:=WObj0;
MoveL [[1554.77,-443,-508.35],[0.032971,0.999448,0.003972,-0.00071],[0,-1,-1,0],[0,9E9,9E9,9E9,9E9,9E9]],Work,z10,custom_tool1\WObj:=WObj0;
MoveL [[1559.94,-442.91,-508.36],[0.032971,0.999448,0.003972,-0.00071],[0,-1,-1,0],[0,9E9,9E9,9E9,9E9,9E9]],Work,z10,custom_tool1\WObj:=WObj0;
MoveL [[1565.11,-442.83,-508.37],[0.032971,0.999448,0.003972,-0.00071],[0,-1,-1,0],[0,9E9,9E9,9E9,9E9,9E9]],Work,z10,custom_tool1\WObj:=WObj0;
MoveL [[1570.27,-442.74,-508.38],[0.032971,0.999448,0.003972,-0.00071],[0,-1,-1,0],[0,9E9,9E9,9E9,9E9,9E9]],Work,z10,custom_tool1\WObj:=WObj0;
MoveL [[1575.44,-442.66,-508.39],[0.032971,0.999448,0.003972,-0.00071],[0,-1,-1,0],[0,9E9,9E9,9E9,9E9,9E9]],Work,z10,custom_tool1\WObj:=WObj0;
MoveL [[1580.6,-442.57,-508.41],[0.032971,0.999448,0.003972,-0.00071],[0,-1,-1,0],[0,9E9,9E9,9E9,9E9,9E9]],Work,z10,custom_tool1\WObj:=WObj0;
MoveL [[1585.77,-442.49,-508.42],[0.032971,0.999448,0.003972,-0.00071],[0,-1,-1,0],[0,9E9,9E9,9E9,9E9,9E9]],Work,z10,custom_tool1\WObj:=WObj0;
MoveL [[1590.94,-442.4,-508.43],[0.032971,0.999448,0.003972,-0.00071],[0,-1,-1,0],[0,9E9,9E9,9E9,9E9,9E9]],Work,z10,custom_tool1\WObj:=WObj0;
MoveL [[1596.1,-442.32,-508.44],[0.032971,0.999448,0.003972,-0.00071],[0,-1,-1,0],[0,9E9,9E9,9E9,9E9,9E9]],Work,z10,custom_tool1\WObj:=WObj0;
MoveL [[1596.1,-442.32,-508.44],[0.032971,0.999448,0.003972,-0.00071],[0,-1,-1,0],[0,9E9,9E9,9E9,9E9,9E9]],Work,fine,custom_tool1\WObj:=WObj0;
SetDo Local_IO_0_DO2,0;
MoveL [[1596.1,-442.32,-478.44],[0.032971,0.999448,0.003972,-0.00071],[0,-1,-1,0],[0,9E9,9E9,9E9,9E9,9E9]],Work,fine,custom_tool1\WObj:=WObj0;
ENDPROC
ENDMODULE

--- Controller Data/v2600-510970_CAADRIA/SYSPAR/EIO.cfg ---
EIO:CFG_1.0:6:1::
#
ETHERNETIP_DEVICE:

      -Name "Local_IO" -VendorName "ABB Robotics" -ProductName "DSQC1030"\
      -Label "ABB Local I/O Device" -Address "192.168.125.100" -VendorId 75\
      -ProductCode 29 -DeviceType 12 -OutputAssembly 100 -InputAssembly 101\
      -ConfigurationAssembly 102 -InputConnectionType "POINT2POINT"\
      -ConnectionPriority "SCHEDULE" -OutputSize 2 -InputSize 2\
      -ConfigurationSize 8\
      -ConfigurationData00 "01 02 09 10 01 08 10 01 00 00 00 00 00 00 00 00"\
      -O2T_RPI 40000 -T2O_RPI 40000
#
EIO_SIGNAL:

      -Name "Local_IO_0_DO1" -SignalType "DO" -Device "Local_IO" -DeviceMap "0"

      -Name "Local_IO_0_DO2" -SignalType "DO" -Device "Local_IO" -DeviceMap "1"

      -Name "Local_IO_0_DO3" -SignalType "DO" -Device "Local_IO" -DeviceMap "2"

      -Name "Local_IO_0_DO4" -SignalType "DO" -Device "Local_IO" -DeviceMap "3"

      -Name "Local_IO_0_DO5" -SignalType "DO" -Device "Local_IO" -DeviceMap "4"

      -Name "Local_IO_0_DO6" -SignalType "DO" -Device "Local_IO" -DeviceMap "5"

      -Name "Local_IO_0_DO7" -SignalType "DO" -Device "Local_IO" -DeviceMap "6"

      -Name "Local_IO_0_DO8" -SignalType "DO" -Device "Local_IO" -DeviceMap "7"

      -Name "Local_IO_0_DO9" -SignalType "DO" -Device "Local_IO" -DeviceMap "8"

      -Name "Local_IO_0_DO10" -SignalType "DO" -Device "Local_IO" -DeviceMap "9"

      -Name "Local_IO_0_DO11" -SignalType "DO" -Device "Local_IO"\
      -DeviceMap "10"

      -Name "Local_IO_0_DO12" -SignalType "DO" -Device "Local_IO"\
      -DeviceMap "11"

      -Name "Local_IO_0_DO13" -SignalType "DO" -Device "Local_IO"\
      -DeviceMap "12"

      -Name "Local_IO_0_DO14" -SignalType "DO" -Device "Local_IO"\
      -DeviceMap "13"

      -Name "Local_IO_0_DO15" -SignalType "DO" -Device "Local_IO"\
      -DeviceMap "14"

      -Name "Local_IO_0_DO16" -SignalType "DO" -Device "Local_IO"\
      -DeviceMap "15"

      -Name "Local_IO_0_DI1" -SignalType "DI" -Device "Local_IO" -DeviceMap "0"

      -Name "Local_IO_0_DI2" -SignalType "DI" -Device "Local_IO" -DeviceMap "1"

      -Name "Local_IO_0_DI3" -SignalType "DI" -Device "Local_IO" -DeviceMap "2"

      -Name "Local_IO_0_DI4" -SignalType "DI" -Device "Local_IO" -DeviceMap "3"

      -Name "Local_IO_0_DI5" -SignalType "DI" -Device "Local_IO" -DeviceMap "4"

      -Name "Local_IO_0_DI6" -SignalType "DI" -Device "Local_IO" -DeviceMap "5"

      -Name "Local_IO_0_DI7" -SignalType "DI" -Device "Local_IO" -DeviceMap "6"

      -Name "Local_IO_0_DI8" -SignalType "DI" -Device "Local_IO" -DeviceMap "7"

      -Name "Local_IO_0_DI9" -SignalType "DI" -Device "Local_IO" -DeviceMap "8"

      -Name "Local_IO_0_DI10" -SignalType "DI" -Device "Local_IO" -DeviceMap "9"

      -Name "Local_IO_0_DI11" -SignalType "DI" -Device "Local_IO"\
      -DeviceMap "10"

      -Name "Local_IO_0_DI12" -SignalType "DI" -Device "Local_IO"\
      -DeviceMap "11"

      -Name "Local_IO_0_DI13" -SignalType "DI" -Device "Local_IO"\
      -DeviceMap "12"

      -Name "Local_IO_0_DI14" -SignalType "DI" -Device "Local_IO"\
      -DeviceMap "13"

      -Name "Local_IO_0_DI15" -SignalType "DI" -Device "Local_IO"\
      -DeviceMap "14"

      -Name "Local_IO_0_DI16" -SignalType "DI" -Device "Local_IO"\
      -DeviceMap "15"
